// TIA Portal V17 export
// export: Created 2023-12-22T15:05:28.4476244Z, ExportSetting WithDefaults, DisplayName Totally Integrated Automation Portal, DisplayVersion V17, DisplayName TIA Portal Openness, DisplayVersion V17, DisplayName TIA Portal Version Control Interface, DisplayVersion V17, DisplayName STEP 7 Professional, DisplayVersion V17, DisplayName STEP 7 Safety, DisplayVersion V17, DisplayName WinCC Advanced, DisplayVersion V17
FUNCTION_BLOCK "DIx_1"   // FB200, LAD
{ S7_Optimized_Access := 'FALSE' }
VERSION : 0.1
// Input - входной сигнал контроллера
// pulse - частота фильтрации дребезга
// Signal - обработанный и отфильтрованный сигнал, используемый в дальнейшем
// stored: AutoNumber false, IsIECCheckEnabled false, SetENOAutomatically false, UDAEnableTagReadback false
   VAR
      AllBlock { S7_SetPoint := 'True'} : "DI_ex";   // Аварийный останов / 2.4 разрешение на работу
      EZ_1_FB_AHLS { S7_SetPoint := 'True'} : "DI_ex";   // Электролизер 1 (Переполнение поддона) / 2.3 Нижний уровень
      Gas_Chanel_1_1 { S7_SetPoint := 'True'} : "DI_ex";   // Загазованность канал 1 (Порог 1) / Ротаметр 1
      Gas_Chanel_1_2 { S7_SetPoint := 'True'} : "DI_ex";   // Загазованность канал 1 (Порог 2) / Ротаметр 2
      Gas_Chanel_2_1 { S7_SetPoint := 'True'} : "DI_ex";   // Загазованность канал 2 (Порог 1) / Ротаметр 3
      Gas_Chanel_2_2 { S7_SetPoint := 'True'} : "DI_ex";   // Загазованность канал 2 (Порог 2) / Датчик переливва
      ALS_1 { S7_SetPoint := 'True'} : "DI_ex";   // Аварийный уровень 1 / Датчик переливва
      KC_1 { S7_SetPoint := 'True'} : "DI_ex";   // Блок клапанов (Сигнал 1)
      KC_2 { S7_SetPoint := 'True'} : "DI_ex";   // Блок клапанов (Сигнал 2)
      signal_10 { S7_SetPoint := 'True'} : "DI_ex";
      signal_11 { S7_SetPoint := 'True'} : "DI_ex";
      signal_12 { S7_SetPoint := 'True'} : "DI_ex";
      signal_13 { S7_SetPoint := 'True'} : "DI_ex";
   END_VAR
   VAR DB_SPECIFIC
      Time_DTL { S7_SetPoint := 'True'} : DTL;
   END_VAR
   // AllBlock.ADDR_Byte := 1;
   // AllBlock.ADDR_Bit := 5;
   // EZ_1_FB_AHLS.ADDR_Byte := 0;
   // EZ_1_FB_AHLS.ADDR_Bit := 2;
   // Gas_Chanel_1_1.ADDR_Bit := 7;
   // Gas_Chanel_1_2.ADDR_Byte := 1;
   // Gas_Chanel_1_2.ADDR_Bit := 0;
   // Gas_Chanel_2_1.ADDR_Byte := 1;
   // Gas_Chanel_2_1.ADDR_Bit := 1;
   // Gas_Chanel_2_2.ADDR_Byte := 1;
   // Gas_Chanel_2_2.ADDR_Bit := 2;
   // ALS_1.ADDR_Byte := 2;
   // ALS_1.ADDR_Bit := 0;
   // KC_1.ADDR_Byte := 1;
   // KC_1.ADDR_Bit := 3;
   // KC_2.ADDR_Byte := 1;
   // KC_2.ADDR_Bit := 4;
   VAR_TEMP   // added for the SCL form of the ladder/FBD networks
      _w1 : Bool;
      _w2 : Bool;
   END_VAR
BEGIN

REGION Network 1: AllBlock
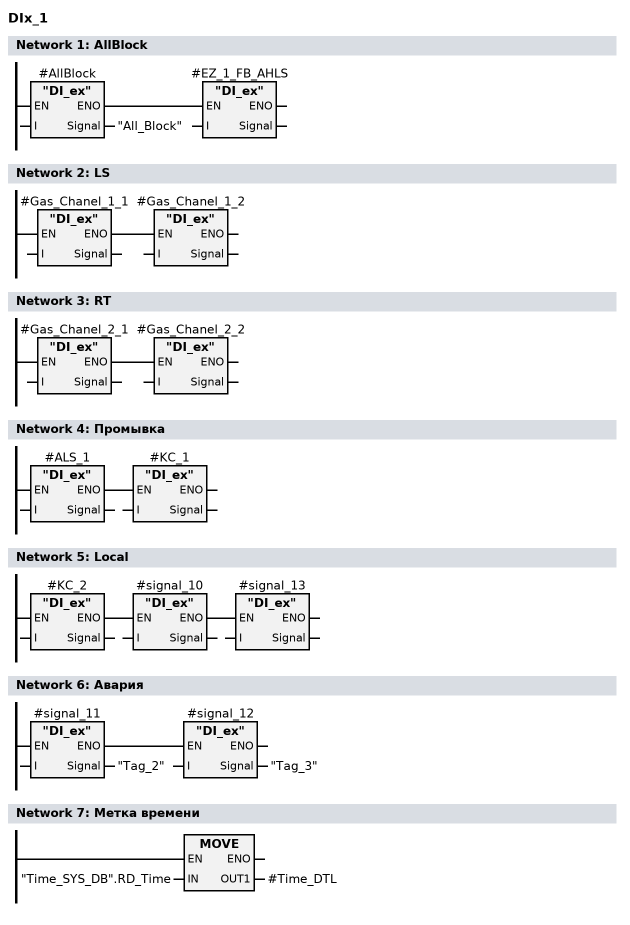
   RUNG wire#powerrail
      #AllBlock(I :=, Signal => "All_Block")
      #EZ_1_FB_AHLS(I :=, Signal =>)
   END_RUNG
   // the same network as SCL:
   #AllBlock(Signal => "All_Block", ENO => #_w1);   // "DI_ex"
   IF #_w1 THEN
       #EZ_1_FB_AHLS();   // "DI_ex"
   END_IF;
END_REGION

REGION Network 2: LS
   RUNG wire#powerrail
      #Gas_Chanel_1_1(I :=, Signal =>)
      #Gas_Chanel_1_2(I :=, Signal =>)
   END_RUNG
   // the same network as SCL:
   #Gas_Chanel_1_1(ENO => #_w1);   // "DI_ex"
   IF #_w1 THEN
       #Gas_Chanel_1_2();   // "DI_ex"
   END_IF;
END_REGION

REGION Network 3: RT
   RUNG wire#powerrail
      #Gas_Chanel_2_1(I :=, Signal =>)
      #Gas_Chanel_2_2(I :=, Signal =>)
   END_RUNG
   // the same network as SCL:
   #Gas_Chanel_2_1(ENO => #_w1);   // "DI_ex"
   IF #_w1 THEN
       #Gas_Chanel_2_2();   // "DI_ex"
   END_IF;
END_REGION

REGION Network 4: Промывка
   RUNG wire#powerrail
      #ALS_1(I :=, Signal =>)
      #KC_1(I :=, Signal =>)
   END_RUNG
   // the same network as SCL:
   #ALS_1(ENO => #_w1);   // "DI_ex"
   IF #_w1 THEN
       #KC_1();   // "DI_ex"
   END_IF;
END_REGION

REGION Network 5: Local
   RUNG wire#powerrail
      #KC_2(I :=, Signal =>)
      #signal_10(I :=, Signal =>)
      #signal_13(I :=, Signal =>)
   END_RUNG
   // the same network as SCL:
   #KC_2(ENO => #_w1);   // "DI_ex"
   #signal_10(EN := #_w1, ENO => #_w2);   // "DI_ex"
   IF #_w2 THEN
       #signal_13();   // "DI_ex"
   END_IF;
END_REGION

REGION Network 6: Авария
   RUNG wire#powerrail
      #signal_11(I :=, Signal => "Tag_2")
      #signal_12(I :=, Signal => "Tag_3")
   END_RUNG
   // the same network as SCL:
   #signal_11(Signal => "Tag_2", ENO => #_w1);   // "DI_ex"
   IF #_w1 THEN
       #signal_12(Signal => "Tag_3");   // "DI_ex"
   END_IF;
END_REGION

REGION Network 7: Метка времени
   RUNG wire#powerrail
      Move(in := "Time_SYS_DB".RD_Time, out1 => #Time_DTL)
   END_RUNG
   // the same network as SCL:
   #Time_DTL := "Time_SYS_DB".RD_Time;
END_REGION
END_FUNCTION_BLOCK
